// TIA Portal V19 export
FUNCTION "AO SCALING" : Void   // FC17, LAD
{ S7_Optimized_Access := 'TRUE' }
// stored: SetENOAutomatically false
   VAR_TEMP   // added for the SCL form of the ladder/FBD networks
      _w1 : Bool;
   END_VAR
BEGIN

REGION Network 1: VFD P-502A
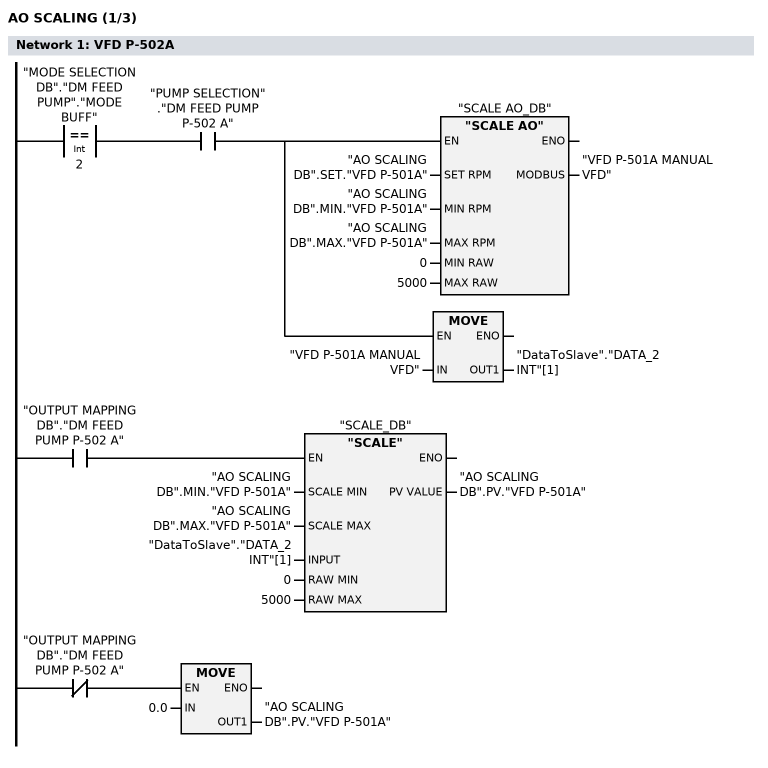
   RUNG wire#powerrail
      { S7_Templates := "SrcType := Int" } EQ_Contact(in1 := "MODE SELECTION DB"."DM FEED PUMP"."MODE BUFF", in2 := 2)
      Contact( "PUMP SELECTION"."DM FEED PUMP P-502 A" )
      wire#w1
      "SCALE AO_DB"("SET RPM" := "AO SCALING DB".SET."VFD P-501A", "MIN RPM" := "AO SCALING DB".MIN."VFD P-501A", "MAX RPM" := "AO SCALING DB".MAX."VFD P-501A", "MIN RAW" := 0, "MAX RAW" := 5000, MODBUS => "VFD P-501A MANUAL VFD")
   END_RUNG
   RUNG wire#w1
      Move(in := "VFD P-501A MANUAL VFD", out1 => "DataToSlave"."DATA_2 INT"[1])
   END_RUNG
   RUNG wire#powerrail
      Contact( "OUTPUT MAPPING DB"."DM FEED PUMP P-502 A" )
      "SCALE_DB"("SCALE MIN" := "AO SCALING DB".MIN."VFD P-501A", "SCALE MAX" := "AO SCALING DB".MAX."VFD P-501A", INPUT := "DataToSlave"."DATA_2 INT"[1], "RAW MIN" := 0, "RAW MAX" := 5000, "PV VALUE" => "AO SCALING DB".PV."VFD P-501A")
   END_RUNG
   RUNG wire#powerrail
      I_Contact( "OUTPUT MAPPING DB"."DM FEED PUMP P-502 A" )
      Move(in := 0.0, out1 => "AO SCALING DB".PV."VFD P-501A")
   END_RUNG
   // the same network as SCL:
   #_w1 := ("MODE SELECTION DB"."DM FEED PUMP"."MODE BUFF" = 2) AND "PUMP SELECTION"."DM FEED PUMP P-502 A";
   IF #_w1 THEN
       "SCALE AO_DB"("SET RPM" := "AO SCALING DB".SET."VFD P-501A",   // "SCALE AO"
                     "MIN RPM" := "AO SCALING DB".MIN."VFD P-501A",
                     "MAX RPM" := "AO SCALING DB".MAX."VFD P-501A",
                     "MIN RAW" := 0,
                     "MAX RAW" := 5000,
                     MODBUS => "VFD P-501A MANUAL VFD");
       "DataToSlave"."DATA_2 INT"[1] := "VFD P-501A MANUAL VFD";
   END_IF;
   IF "OUTPUT MAPPING DB"."DM FEED PUMP P-502 A" THEN
       "SCALE_DB"("SCALE MIN" := "AO SCALING DB".MIN."VFD P-501A",   // "SCALE"
                  "SCALE MAX" := "AO SCALING DB".MAX."VFD P-501A",
                  INPUT := "DataToSlave"."DATA_2 INT"[1],
                  "RAW MIN" := 0,
                  "RAW MAX" := 5000,
                  "PV VALUE" => "AO SCALING DB".PV."VFD P-501A");
   END_IF;
   IF NOT "OUTPUT MAPPING DB"."DM FEED PUMP P-502 A" THEN "AO SCALING DB".PV."VFD P-501A" := 0.0; END_IF;
END_REGION

REGION Network 2: VFD P-502B
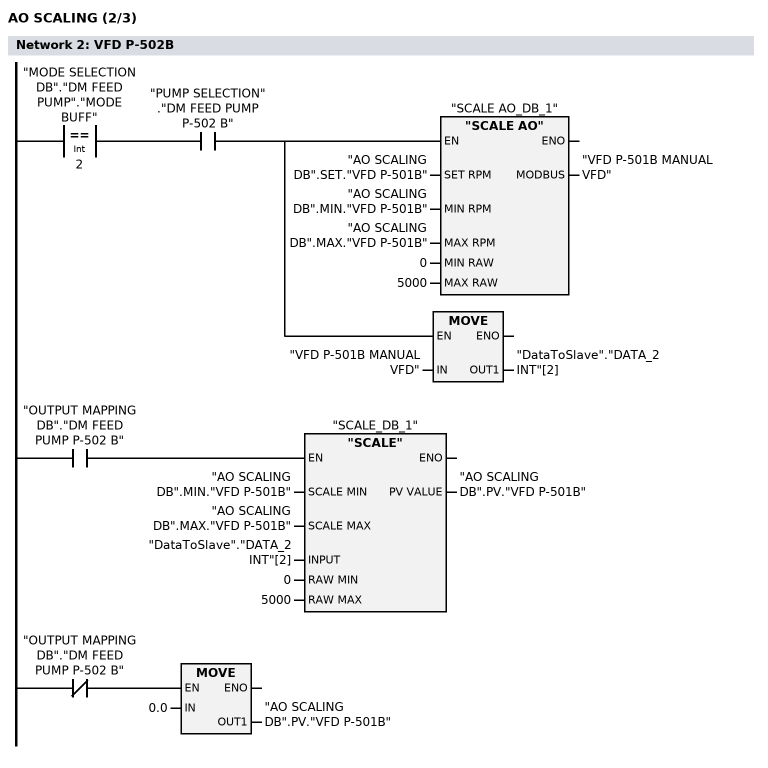
   RUNG wire#powerrail
      { S7_Templates := "SrcType := Int" } EQ_Contact(in1 := "MODE SELECTION DB"."DM FEED PUMP"."MODE BUFF", in2 := 2)
      Contact( "PUMP SELECTION"."DM FEED PUMP P-502 B" )
      wire#w1
      "SCALE AO_DB_1"("SET RPM" := "AO SCALING DB".SET."VFD P-501B", "MIN RPM" := "AO SCALING DB".MIN."VFD P-501B", "MAX RPM" := "AO SCALING DB".MAX."VFD P-501B", "MIN RAW" := 0, "MAX RAW" := 5000, MODBUS => "VFD P-501B MANUAL VFD")
   END_RUNG
   RUNG wire#w1
      Move(in := "VFD P-501B MANUAL VFD", out1 => "DataToSlave"."DATA_2 INT"[2])
   END_RUNG
   RUNG wire#powerrail
      Contact( "OUTPUT MAPPING DB"."DM FEED PUMP P-502 B" )
      "SCALE_DB_1"("SCALE MIN" := "AO SCALING DB".MIN."VFD P-501B", "SCALE MAX" := "AO SCALING DB".MAX."VFD P-501B", INPUT := "DataToSlave"."DATA_2 INT"[2], "RAW MIN" := 0, "RAW MAX" := 5000, "PV VALUE" => "AO SCALING DB".PV."VFD P-501B")
   END_RUNG
   RUNG wire#powerrail
      I_Contact( "OUTPUT MAPPING DB"."DM FEED PUMP P-502 B" )
      Move(in := 0.0, out1 => "AO SCALING DB".PV."VFD P-501B")
   END_RUNG
   // the same network as SCL:
   #_w1 := ("MODE SELECTION DB"."DM FEED PUMP"."MODE BUFF" = 2) AND "PUMP SELECTION"."DM FEED PUMP P-502 B";
   IF #_w1 THEN
       "SCALE AO_DB_1"("SET RPM" := "AO SCALING DB".SET."VFD P-501B",   // "SCALE AO"
                       "MIN RPM" := "AO SCALING DB".MIN."VFD P-501B",
                       "MAX RPM" := "AO SCALING DB".MAX."VFD P-501B",
                       "MIN RAW" := 0,
                       "MAX RAW" := 5000,
                       MODBUS => "VFD P-501B MANUAL VFD");
       "DataToSlave"."DATA_2 INT"[2] := "VFD P-501B MANUAL VFD";
   END_IF;
   IF "OUTPUT MAPPING DB"."DM FEED PUMP P-502 B" THEN
       "SCALE_DB_1"("SCALE MIN" := "AO SCALING DB".MIN."VFD P-501B",   // "SCALE"
                    "SCALE MAX" := "AO SCALING DB".MAX."VFD P-501B",
                    INPUT := "DataToSlave"."DATA_2 INT"[2],
                    "RAW MIN" := 0,
                    "RAW MAX" := 5000,
                    "PV VALUE" => "AO SCALING DB".PV."VFD P-501B");
   END_IF;
   IF NOT "OUTPUT MAPPING DB"."DM FEED PUMP P-502 B" THEN "AO SCALING DB".PV."VFD P-501B" := 0.0; END_IF;
END_REGION

REGION Network 3: VFD P-502C
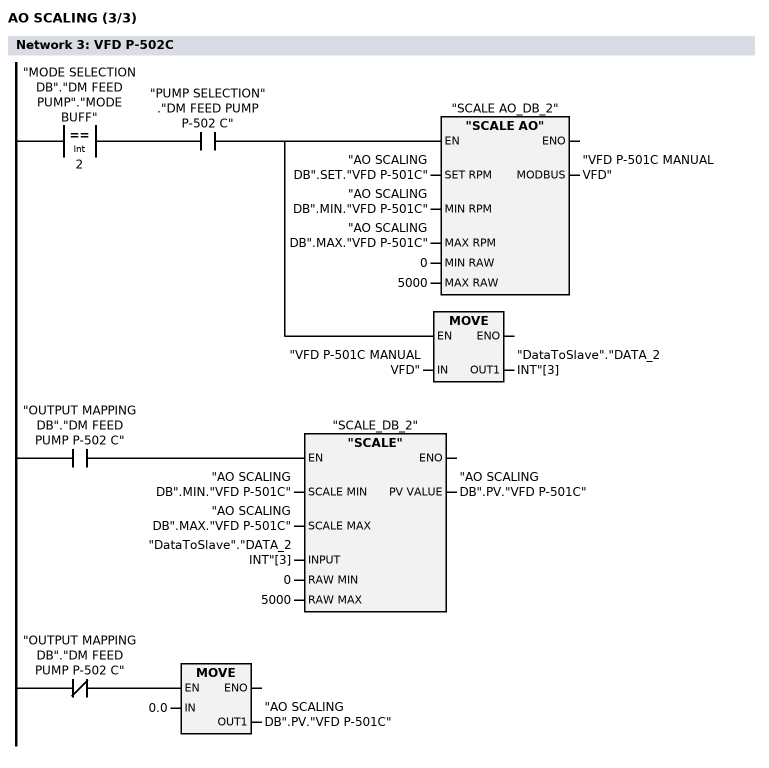
   RUNG wire#powerrail
      { S7_Templates := "SrcType := Int" } EQ_Contact(in1 := "MODE SELECTION DB"."DM FEED PUMP"."MODE BUFF", in2 := 2)
      Contact( "PUMP SELECTION"."DM FEED PUMP P-502 C" )
      wire#w1
      "SCALE AO_DB_2"("SET RPM" := "AO SCALING DB".SET."VFD P-501C", "MIN RPM" := "AO SCALING DB".MIN."VFD P-501C", "MAX RPM" := "AO SCALING DB".MAX."VFD P-501C", "MIN RAW" := 0, "MAX RAW" := 5000, MODBUS => "VFD P-501C MANUAL VFD")
   END_RUNG
   RUNG wire#w1
      Move(in := "VFD P-501C MANUAL VFD", out1 => "DataToSlave"."DATA_2 INT"[3])
   END_RUNG
   RUNG wire#powerrail
      Contact( "OUTPUT MAPPING DB"."DM FEED PUMP P-502 C" )
      "SCALE_DB_2"("SCALE MIN" := "AO SCALING DB".MIN."VFD P-501C", "SCALE MAX" := "AO SCALING DB".MAX."VFD P-501C", INPUT := "DataToSlave"."DATA_2 INT"[3], "RAW MIN" := 0, "RAW MAX" := 5000, "PV VALUE" => "AO SCALING DB".PV."VFD P-501C")
   END_RUNG
   RUNG wire#powerrail
      I_Contact( "OUTPUT MAPPING DB"."DM FEED PUMP P-502 C" )
      Move(in := 0.0, out1 => "AO SCALING DB".PV."VFD P-501C")
   END_RUNG
   // the same network as SCL:
   #_w1 := ("MODE SELECTION DB"."DM FEED PUMP"."MODE BUFF" = 2) AND "PUMP SELECTION"."DM FEED PUMP P-502 C";
   IF #_w1 THEN
       "SCALE AO_DB_2"("SET RPM" := "AO SCALING DB".SET."VFD P-501C",   // "SCALE AO"
                       "MIN RPM" := "AO SCALING DB".MIN."VFD P-501C",
                       "MAX RPM" := "AO SCALING DB".MAX."VFD P-501C",
                       "MIN RAW" := 0,
                       "MAX RAW" := 5000,
                       MODBUS => "VFD P-501C MANUAL VFD");
       "DataToSlave"."DATA_2 INT"[3] := "VFD P-501C MANUAL VFD";
   END_IF;
   IF "OUTPUT MAPPING DB"."DM FEED PUMP P-502 C" THEN
       "SCALE_DB_2"("SCALE MIN" := "AO SCALING DB".MIN."VFD P-501C",   // "SCALE"
                    "SCALE MAX" := "AO SCALING DB".MAX."VFD P-501C",
                    INPUT := "DataToSlave"."DATA_2 INT"[3],
                    "RAW MIN" := 0,
                    "RAW MAX" := 5000,
                    "PV VALUE" => "AO SCALING DB".PV."VFD P-501C");
   END_IF;
   IF NOT "OUTPUT MAPPING DB"."DM FEED PUMP P-502 C" THEN "AO SCALING DB".PV."VFD P-501C" := 0.0; END_IF;
END_REGION
END_FUNCTION
